// TwinCAT 3 PLC project AdsGo_Test
// ProgramVersion: 3.1.4026.21
// libraries:
//   Tc2_Standard, * (Beckhoff Automation GmbH)
//   Tc2_System, * (Beckhoff Automation GmbH)
//   Tc3_Module, * (Beckhoff Automation GmbH)
// project tree:
//   Lib/ TestStruct.TcDUT
//   Globals/ Global.TcGVL (not stored)
//   Programs/ Main.TcPOU
//   Tasks/ PlcTask.TcTTO
// real-time tasks:
//   TASK 2ms: cycle T#2ms, priority 3, ADS port 350
//   TASK 10ms: cycle T#10ms, priority 4, ADS port 351
//   TASK 200ms: cycle T#200000us, priority 6, ADS port 352
//   TASK FileWriterTask: cycle T#200000us, priority 1, ADS port 353
//   TASK PlcTask: cycle T#10ms, priority 20, ADS port 354

CONFIGURATION AdsGo_Test
    RESOURCE PLC ON TwinCAT3
        TASK PlcTask(INTERVAL := T#10ms, PRIORITY := 20);
        PROGRAM Main WITH PlcTask : Main;
    END_RESOURCE
END_CONFIGURATION

// ---- Lib/TestStruct.TcDUT
TYPE TestStruct :
STRUCT
	counter : INT;
	ready : BOOL;
	int_array : ARRAY[0..50] OF INT;  
END_STRUCT
END_TYPE

// ---- Programs/Main.TcPOU
PROGRAM Main
VAR
	timer : Ton;
	tick : BOOL;
	
	{attribute 'displaymode':='hex'} 
    var_with_standard_attribute : DWORD;
	
	{attribute 'my_custom_attribute'}
	var_with_custom_attribute : STRING(255) := 'I have attribute {attribute $'my_custom_attribute$'}';
END_VAR

// ------------------------------------------------------------
// A) Cycle-based behavior (each PLC scan)
// ------------------------------------------------------------

IF Global.int_counter_active THEN
    Global.int_counter := Global.int_counter + 1;
END_IF

IF Global.bool_toggle_active THEN
    Global.bool_toggle := NOT Global.bool_toggle;
END_IF

// ------------------------------------------------------------
// B) Time-based behavior (every Global.cycle_period)
// This triggers a `tick` each time the Ton timer elapses.
// ------------------------------------------------------------
timer(IN := TRUE, PT := Global.cycle_period);

// bTick is TRUE only when timer is done
tick := timer.Q;

IF tick THEN
    // Do the same actions, but only on the tick
    IF Global.timed_int_counter_active THEN
        Global.timer_int_counter := Global.timer_int_counter + 1;
    END_IF

    IF Global.timed_bool_toggle_active THEN
        Global.timed_bool_toggle := NOT Global.timed_bool_toggle;
    END_IF

    // Retrigger timer (create a periodic pulse)
    timer(IN := FALSE);
END_IF

END_PROGRAM
